FUNCTION_BLOCK ADI_TO_AW (* Composite FB for converting ADI (DINT) adapter to AW (WORD) adapter *)
  (* Standard: 61499-2; Description: Copyright (c) 2026 HR Agrartechnik GmbH This program and the accompanying materials are made available under the terms of the Eclipse Public License 2.0 which is available at https://www.eclipse.org/legal/epl-2.0/ SPDX-License-Identifier: EPL-2.0 *)
  (* Version 1.0, 2026-02-17, Franz Höpfinger, HR Agrartechnik GmbH *)
  PACKAGE adapter::conversion::unidirectional;
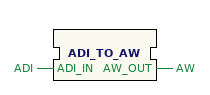
  SOCKETS
    ADI_IN : adapter::types::unidirectional::ADI; (* DINT Adapter Input *)
  END_SOCKETS
  PLUGS
    AW_OUT : adapter::types::unidirectional::AW; (* WORD Adapter Output *)
  END_PLUGS
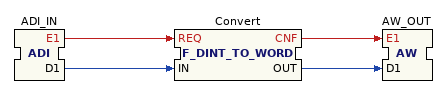
  FBS
    Convert : iec61131::conversion::F_DINT_TO_WORD;
  END_FBS
  EVENT_CONNECTIONS
    ADI_IN.E1 TO Convert.REQ;
    Convert.CNF TO AW_OUT.E1;
  END_CONNECTIONS
  DATA_CONNECTIONS
    ADI_IN.D1 TO Convert.IN;
    Convert.OUT TO AW_OUT.D1;
  END_CONNECTIONS
END_FUNCTION_BLOCK
